{attribute 'pack_mode' := '1'}
TYPE ST_ReadListDataArrayInt :
STRUCT
	stReadListReturnInfo	: ARRAY [1..gNodeIDCount_Array] OF ST_UAReadListReturnInfo; // must be less than nMaxNodeIDsInList, nMaxNodeIDsInList = 10
	nArrIntVar1				: ARRAY [1..10] OF INT; 
	nArrDintVar2			: ARRAY [1..2] OF DINT; 	
END_STRUCT
END_TYPE

(* stored: Version 1.1.0.1, ProductVersion 3.1.4022.6
   DUT ST_ReadListDataArrayInt: Id {2fb3ff15-8f83-42fe-bd03-3967d32958e1} *)
